(* PLC project Doqu_ges.project, CODESYS CODESYS V3.5 SP20 Patch 1 *)
(* stored: creationDateTime 2024-07-29T14:44:46.2377894, modificationDateTime 2024-07-20T22:10:28.0263958 *)

{attribute 'qualified_only'}
VAR_GLOBAL  (* GVL_1 *)
  Pry_Net_Radition_104 AT %QD10 : REAL;  (* NEW Pyronometer *)
  Pry_Compensated_Radition_104 AT %QD11 : REAL;
  Pry_Temp_104 AT %QD12 : REAL;
  Pry_External_Voltage_104 AT %QD13 : REAL;
  Refcel1_Net_Radition_104 AT %QD14 : REAL;  (* Refcel-1 *)
  Refcel1_Compensated_Radition_104 AT %QD15 : REAL;
  Refcel1_Temp_104 AT %QD16 : REAL;
  Refcel2_Net_Radition_104 AT %QD17 : REAL;  (* Refcel-2 *)
  Refcel2_Compensated_Radition_104 AT %QD18 : REAL;
  Refcel2_Temp_104 AT %QD19 : REAL;
  H1_Ia_104 AT %QD20 : REAL;  (* H1_Relay *)
  H1_Ib_104 AT %QD21 : REAL;
  H1_Ic_104 AT %QD22 : REAL;
  H1_Fault_Ia_104 AT %QD23 : REAL;
  H1_Fault_Ib_104 AT %QD24 : REAL;
  H1_Fault_Ic_104 AT %QD25 : REAL;
  H1_In_104 AT %QD26 : REAL;
  H1_Va_104 AT %QD27 : REAL;
  H1_Vb_104 AT %QD28 : REAL;
  H1_Vc_104 AT %QD29 : REAL;
  H1_Van_104 AT %QD30 : REAL;
  H1_Vbn_104 AT %QD31 : REAL;
  H1_Vcn_104 AT %QD32 : REAL;
  H1_F_104 AT %QD33 : REAL;
  H1_THD_Ia_104 AT %QD34 : REAL;
  H1_THD_Ib_104 AT %QD35 : REAL;
  H1_THD_Ic_104 AT %QD36 : REAL;
  H1_THD_Va_104 AT %QD37 : REAL;
  H1_THD_Vb_104 AT %QD38 : REAL;
  H1_THD_Vc_104 AT %QD39 : REAL;
  H1_Pf_104 AT %QD40 : REAL;
  H1_P_104 AT %QD41 : REAL;
  H1_Q_104 AT %QD42 : REAL;
  H1_S_104 AT %QD43 : REAL;
  H1_Wpneg_104 AT %QD44 : REAL;
  H1_Wqneg_104 AT %QD45 : REAL;
  H1_Wppos_104 AT %QD46 : REAL;
  H1_Wqpos_104 AT %QD47 : REAL;
  H1_CB_State_104 AT %QD48 : REAL;
  H1_DS_State_104 AT %QD49 : REAL;
  H1_EDS_State_104 AT %QD50 : REAL;
  H1_Remote_State_104 AT %QD51 : REAL;
  H1_OC_State1_104 AT %QD52 : REAL;
  H1_OC_State2_104 AT %QD53 : REAL;
  H1_EOC_State1_104 AT %QD54 : REAL;
  H1_EOC_State2_104 AT %QD55 : REAL;
  H1_Relay_Fault_104 AT %QD56 : REAL;
  H2_Ia_104 AT %QD57 : REAL;  (* H2_ION *)
  H2_Ib_104 AT %QD58 : REAL;
  H2_Ic_104 AT %QD59 : REAL;
  H2_Van_104 AT %QD60 : REAL;
  H2_Vbn_104 AT %QD61 : REAL;
  H2_Vcn_104 AT %QD62 : REAL;
  H2_Vab_104 AT %QD63 : REAL;
  H2_Vbc_104 AT %QD64 : REAL;
  H2_Vac_104 AT %QD65 : REAL;
  H2_F_104 AT %QD66 : REAL;
  H2_PF_104 AT %QD67 : REAL;
  H2_THDIA_104 AT %QD68 : REAL;
  H2_THDIB_104 AT %QD69 : REAL;
  H2_THDIC_104 AT %QD70 : REAL;
  H2_THDVA_104 AT %QD71 : REAL;
  H2_THDVB_104 AT %QD72 : REAL;
  H2_THDVC_104 AT %QD73 : REAL;
  H2_P_104 AT %QD74 : REAL;
  H2_Q_104 AT %QD75 : REAL;
  H2_S_104 AT %QD76 : REAL;
  H2_Wppos_104 AT %QD77 : REAL;
  H2_Wpneg_104 AT %QD78 : REAL;
  H2_Wqpos_104 AT %QD79 : REAL;
  H2_Wqneg_104 AT %QD80 : REAL;
  H2_Ia_Angle_104 AT %QD81 : REAL;
  H2_Ib_Angle_104 AT %QD82 : REAL;
  H2_Ic_Angle_104 AT %QD83 : REAL;
  H2_Va_Angle_104 AT %QD84 : REAL;
  H2_Vb_Angle_104 AT %QD85 : REAL;
  H2_Vc_Angle_104 AT %QD86 : REAL;
  H2_V1Plt_104 AT %QD87 : REAL;
  H2_V1Pst_104 AT %QD88 : REAL;
  H2_V2Plt_104 AT %QD89 : REAL;
  H2_V2Pst_104 AT %QD90 : REAL;
  H2_V3Plt_104 AT %QD91 : REAL;
  H2_V3Pst_104 AT %QD92 : REAL;
  INV1_Status_104 AT %QD93 : REAL;  (* *Inverter-1 *)
  INV1_Status_1044 : REAL;
  INV1_Pin_104 AT %QD94 : REAL;
  INV1_Pv1_voltage_104 AT %QD95 : REAL;
  INV1_Pv1_current_104 AT %QD96 : REAL;
  INV1_Pv1_Pin_104 AT %QD97 : REAL;
  INV1_Pv2_voltage_104 AT %QD98 : REAL;
  INV1_Pv2_current_104 AT %QD99 : REAL;
  INV1_Pv2_Pin_104 AT %QD100 : REAL;
  INV1_Pv3_voltage_104 AT %QD101 : REAL;
  INV1_Pv3_current_104 AT %QD102 : REAL;
  INV1_Pv3_Pin_104 AT %QD103 : REAL;
  INV1_Pv4_voltage_104 AT %QD104 : REAL;
  INV1_Pv4_current_104 AT %QD105 : REAL;
  INV1_Pv4_Pin_104 AT %QD106 : REAL;
  INV1_Pv5_voltage_104 AT %QD107 : REAL;
  INV1_Pv5_current_104 AT %QD108 : REAL;
  INV1_Pv5_Pin_104 AT %QD109 : REAL;
  INV1_Pv6_voltage_104 AT %QD110 : REAL;
  INV1_Pv6_current_104 AT %QD111 : REAL;
  INV1_Pv6_Pin_104 AT %QD112 : REAL;
  INV1_Pv7_voltage_104 AT %QD113 : REAL;
  INV1_Pv7_current_104 AT %QD114 : REAL;
  INV1_Pv7_Pin_104 AT %QD115 : REAL;
  INV1_Pv8_voltage_104 AT %QD116 : REAL;
  INV1_Pv8_current_104 AT %QD117 : REAL;
  INV1_Pv8_Pin_104 AT %QD118 : REAL;
  INV1_Pv9_voltage_104 AT %QD119 : REAL;
  INV1_Pv9_current_104 AT %QD120 : REAL;
  INV1_Pv9_Pin_104 AT %QD121 : REAL;
  INV1_Pv10_voltage_104 AT %QD122 : REAL;
  INV1_Pv10_current_104 AT %QD123 : REAL;
  INV1_Pv10_Pin_104 AT %QD124 : REAL;
  INV1_Pac_out_104 AT %QD125 : REAL;
  INV1_Fac_104 AT %QD126 : REAL;
  INV1_Vac1_104 AT %QD127 : REAL;
  INV1_Iac1_104 AT %QD128 : REAL;
  INV1_Pac1_104 AT %QD129 : REAL;
  INV1_Vac2_104 AT %QD130 : REAL;
  INV1_Iac2_104 AT %QD131 : REAL;
  INV1_Pac2_104 AT %QD132 : REAL;
  INV1_Vac3_104 AT %QD133 : REAL;
  INV1_Iac3_104 AT %QD134 : REAL;
  INV1_Pac3_104 AT %QD135 : REAL;
  INV1_Vac_RS_104 AT %QD136 : REAL;
  INV1_Vac_ST_104 AT %QD137 : REAL;
  INV1_Vac_TR_104 AT %QD138 : REAL;
  INV1_Eactoday_104 AT %QD139 : REAL;
  INV1_Eactotal_104 AT %QD140 : REAL;
  INV1_Timetotal_104 AT %QD141 : REAL;
  INV1_Epv1_today_104 AT %QD142 : REAL;
  INV1_Epv1_total_104 AT %QD143 : REAL;
  INV1_Epv2_today_104 AT %QD144 : REAL;
  INV1_Epv2_total_104 AT %QD145 : REAL;
  INV1_Epv3_today_104 AT %QD146 : REAL;
  INV1_Epv3_total_104 AT %QD147 : REAL;
  INV1_Epv4_today_104 AT %QD148 : REAL;
  INV1_Epv4_total_104 AT %QD149 : REAL;
  INV1_Epv5_today_104 AT %QD150 : REAL;
  INV1_Epv5_total_104 AT %QD151 : REAL;
  INV1_Epv6_today_104 AT %QD152 : REAL;
  INV1_Epv6_total_104 AT %QD153 : REAL;
  INV1_Epv7_today_104 AT %QD154 : REAL;
  INV1_Epv7_total_104 AT %QD155 : REAL;
  INV1_Epv8_today_104 AT %QD156 : REAL;
  INV1_Epv8_total_104 AT %QD157 : REAL;
  INV1_Epv9_today_104 AT %QD158 : REAL;
  INV1_Epv9_total_104 AT %QD159 : REAL;
  INV1_Epv10_today_104 AT %QD160 : REAL;
  INV1_Epv10_total_104 AT %QD161 : REAL;
  INV1_Epv_total_104 AT %QD162 : REAL;
  INV1_Temp1_104 AT %QD163 : REAL;
  INV1_Temp2_104 AT %QD164 : REAL;
  INV1_Temp3_104 AT %QD165 : REAL;
  INV1_Temp4_104 AT %QD166 : REAL;
  INV1_BatVolt_DSP_104 AT %QD167 : REAL;
  INV1_P_Bus_Voltage_104 AT %QD168 : REAL;
  INV1_N_Bus_Voltage_104 AT %QD169 : REAL;
  INV1_IPF_104 AT %QD170 : REAL;
  INV1_String_V1_104 AT %QD171 : REAL;
  INV1_String_I1_104 AT %QD172 : REAL;
  INV1_String_V2_104 AT %QD173 : REAL;
  INV1_String_I2_104 AT %QD174 : REAL;
  INV1_String_V3_104 AT %QD175 : REAL;
  INV1_String_I3_104 AT %QD176 : REAL;
  INV1_String_V4_104 AT %QD177 : REAL;
  INV1_String_I4_104 AT %QD178 : REAL;
  INV1_String_V5_104 AT %QD179 : REAL;
  INV1_String_I5_104 AT %QD180 : REAL;
  INV1_String_V6_104 AT %QD181 : REAL;
  INV1_String_I6_104 AT %QD182 : REAL;
  INV1_String_V7_104 AT %QD183 : REAL;
  INV1_String_I7_104 AT %QD184 : REAL;
  INV1_String_V8_104 AT %QD185 : REAL;
  INV1_String_I8_104 AT %QD186 : REAL;
  INV1_String_V9_104 AT %QD187 : REAL;
  INV1_String_I9_104 AT %QD188 : REAL;
  INV1_String_V10_104 AT %QD189 : REAL;
  INV1_String_I10_104 AT %QD190 : REAL;
  INV1_String_V11_104 AT %QD191 : REAL;
  INV1_String_I11_104 AT %QD192 : REAL;
  INV1_String_V12_104 AT %QD193 : REAL;
  INV1_String_I12_104 AT %QD194 : REAL;
  INV1_String_V13_104 AT %QD195 : REAL;
  INV1_String_I13_104 AT %QD196 : REAL;
  INV1_String_V14_104 AT %QD197 : REAL;
  INV1_String_I14_104 AT %QD198 : REAL;
  INV1_String_V15_104 AT %QD199 : REAL;
  INV1_String_I15_104 AT %QD200 : REAL;
  INV1_String_V16_104 AT %QD201 : REAL;
  INV1_String_I16_104 AT %QD202 : REAL;
  INV1_String_V17_104 AT %QD203 : REAL;
  INV1_String_I17_104 AT %QD204 : REAL;
  INV1_String_V18_104 AT %QD205 : REAL;
  INV1_String_I18_104 AT %QD206 : REAL;
  INV1_String_V19_104 AT %QD207 : REAL;
  INV1_String_I19_104 AT %QD208 : REAL;
  INV1_String_V20_104 AT %QD209 : REAL;
  INV1_String_I20_104 AT %QD210 : REAL;
  INV1_Fan1_Fault_104 AT %QD211 : REAL;
  INV1_Fan2_Fault_104 AT %QD212 : REAL;
  INV1_Fan3_Fault_104 AT %QD213 : REAL;
  INV1_Fan4_Fault_104 AT %QD214 : REAL;
  INV2_Status_104 AT %QD215 : REAL;  (* Inverter-2 *)
  INV2_Pin_104 AT %QD216 : REAL;
  INV2_Pv1_voltage_104 AT %QD217 : REAL;
  INV2_Pv1_current_104 AT %QD218 : REAL;
  INV2_Pv1_Pin_104 AT %QD219 : REAL;
  INV2_Pv2_voltage_104 AT %QD220 : REAL;
  INV2_Pv2_current_104 AT %QD221 : REAL;
  INV2_Pv2_Pin_104 AT %QD222 : REAL;
  INV2_Pv3_voltage_104 AT %QD223 : REAL;
  INV2_Pv3_current_104 AT %QD224 : REAL;
  INV2_Pv3_Pin_104 AT %QD225 : REAL;
  INV2_Pv4_voltage_104 AT %QD226 : REAL;
  INV2_Pv4_current_104 AT %QD227 : REAL;
  INV2_Pv4_Pin_104 AT %QD228 : REAL;
  INV2_Pv5_voltage_104 AT %QD229 : REAL;
  INV2_Pv5_current_104 AT %QD230 : REAL;
  INV2_Pv5_Pin_104 AT %QD231 : REAL;
  INV2_Pv6_voltage_104 AT %QD232 : REAL;
  INV2_Pv6_current_104 AT %QD233 : REAL;
  INV2_Pv6_Pin_104 AT %QD234 : REAL;
  INV2_Pv7_voltage_104 AT %QD235 : REAL;
  INV2_Pv7_current_104 AT %QD236 : REAL;
  INV2_Pv7_Pin_104 AT %QD237 : REAL;
  INV2_Pv8_voltage_104 AT %QD238 : REAL;
  INV2_Pv8_current_104 AT %QD239 : REAL;
  INV2_Pv8_Pin_104 AT %QD240 : REAL;
  INV2_Pv9_voltage_104 AT %QD241 : REAL;
  INV2_Pv9_current_104 AT %QD242 : REAL;
  INV2_Pv9_Pin_104 AT %QD243 : REAL;
  INV2_Pv10_voltage_104 AT %QD244 : REAL;
  INV2_Pv10_current_104 AT %QD245 : REAL;
  INV2_Pv10_Pin_104 AT %QD246 : REAL;
  INV2_Pac_out_104 AT %QD247 : REAL;
  INV2_Fac_104 AT %QD248 : REAL;
  INV2_Vac1_104 AT %QD249 : REAL;
  INV2_Iac1_104 AT %QD250 : REAL;
  INV2_Pac1_104 AT %QD251 : REAL;
  INV2_Vac2_104 AT %QD252 : REAL;
  INV2_Iac2_104 AT %QD253 : REAL;
  INV2_Pac2_104 AT %QD254 : REAL;
  INV2_Vac3_104 AT %QD255 : REAL;
  INV2_Iac3_104 AT %QD256 : REAL;
  INV2_Pac3_104 AT %QD257 : REAL;
  INV2_Vac_RS_104 AT %QD258 : REAL;
  INV2_Vac_ST_104 AT %QD259 : REAL;
  INV2_Vac_TR_104 AT %QD260 : REAL;
  INV2_Eactoday_104 AT %QD261 : REAL;
  INV2_Eactotal_104 AT %QD262 : REAL;
  INV2_Timetotal_104 AT %QD263 : REAL;
  INV2_Epv1_today_104 AT %QD264 : REAL;
  INV2_Epv1_total_104 AT %QD265 : REAL;
  INV2_Epv2_today_104 AT %QD266 : REAL;
  INV2_Epv2_total_104 AT %QD267 : REAL;
  INV2_Epv3_today_104 AT %QD268 : REAL;
  INV2_Epv3_total_104 AT %QD269 : REAL;
  INV2_Epv4_today_104 AT %QD270 : REAL;
  INV2_Epv4_total_104 AT %QD271 : REAL;
  INV2_Epv5_today_104 AT %QD272 : REAL;
  INV2_Epv5_total_104 AT %QD273 : REAL;
  INV2_Epv6_today_104 AT %QD274 : REAL;
  INV2_Epv6_total_104 AT %QD275 : REAL;
  INV2_Epv7_today_104 AT %QD276 : REAL;
  INV2_Epv7_total_104 AT %QD277 : REAL;
  INV2_Epv8_today_104 AT %QD278 : REAL;
  INV2_Epv8_total_104 AT %QD279 : REAL;
  INV2_Epv9_today_104 AT %QD280 : REAL;
  INV2_Epv9_total_104 AT %QD281 : REAL;
  INV2_Epv10_today_104 AT %QD282 : REAL;
  INV2_Epv10_total_104 AT %QD283 : REAL;
  INV2_Epv_total_104 AT %QD284 : REAL;
  INV2_Temp1_104 AT %QD285 : REAL;
  INV2_Temp2_104 AT %QD286 : REAL;
  INV2_Temp3_104 AT %QD287 : REAL;
  INV2_Temp4_104 AT %QD288 : REAL;
  INV2_BatVolt_DSP_104 AT %QD289 : REAL;
  INV2_P_Bus_Voltage_104 AT %QD290 : REAL;
  INV2_N_Bus_Voltage_104 AT %QD291 : REAL;
  INV2_IPF_104 AT %QD292 : REAL;
  INV2_String_V1_104 AT %QD293 : REAL;
  INV2_String_I1_104 AT %QD294 : REAL;
  INV2_String_V2_104 AT %QD295 : REAL;
  INV2_String_I2_104 AT %QD296 : REAL;
  INV2_String_V3_104 AT %QD297 : REAL;
  INV2_String_I3_104 AT %QD298 : REAL;
  INV2_String_V4_104 AT %QD299 : REAL;
  INV2_String_I4_104 AT %QD300 : REAL;
  INV2_String_V5_104 AT %QD301 : REAL;
  INV2_String_I5_104 AT %QD302 : REAL;
  INV2_String_V6_104 AT %QD303 : REAL;
  INV2_String_I6_104 AT %QD304 : REAL;
  INV2_String_V7_104 AT %QD305 : REAL;
  INV2_String_I7_104 AT %QD306 : REAL;
  INV2_String_V8_104 AT %QD307 : REAL;
  INV2_String_I8_104 AT %QD308 : REAL;
  INV2_String_V9_104 AT %QD309 : REAL;
  INV2_String_I9_104 AT %QD310 : REAL;
  INV2_String_V10_104 AT %QD311 : REAL;
  INV2_String_I10_104 AT %QD312 : REAL;
  INV2_String_V11_104 AT %QD313 : REAL;
  INV2_String_I11_104 AT %QD314 : REAL;
  INV2_String_V12_104 AT %QD315 : REAL;
  INV2_String_I12_104 AT %QD316 : REAL;
  INV2_String_V13_104 AT %QD317 : REAL;
  INV2_String_I13_104 AT %QD318 : REAL;
  INV2_String_V14_104 AT %QD319 : REAL;
  INV2_String_I14_104 AT %QD320 : REAL;
  INV2_String_V15_104 AT %QD321 : REAL;
  INV2_String_I15_104 AT %QD322 : REAL;
  INV2_String_V16_104 AT %QD323 : REAL;
  INV2_String_I16_104 AT %QD324 : REAL;
  INV2_String_V17_104 AT %QD325 : REAL;
  INV2_String_I17_104 AT %QD326 : REAL;
  INV2_String_V18_104 AT %QD327 : REAL;
  INV2_String_I18_104 AT %QD328 : REAL;
  INV2_String_V19_104 AT %QD329 : REAL;
  INV2_String_I19_104 AT %QD330 : REAL;
  INV2_String_V20_104 AT %QD331 : REAL;
  INV2_String_I20_104 AT %QD332 : REAL;
  INV2_Fan1_Fault_104 AT %QD333 : REAL;
  INV2_Fan2_Fault_104 AT %QD334 : REAL;
  INV2_Fan3_Fault_104 AT %QD335 : REAL;
  INV2_Fan4_Fault_104 AT %QD336 : REAL;
  INV3_Status_104 AT %QD337 : REAL;  (* *Inverter-3* *)
  INV3_Pin_104 AT %QD338 : REAL;
  INV3_Pv1_voltage_104 AT %QD339 : REAL;
  INV3_Pv1_current_104 AT %QD340 : REAL;
  INV3_Pv1_Pin_104 AT %QD341 : REAL;
  INV3_Pv2_voltage_104 AT %QD342 : REAL;
  INV3_Pv2_current_104 AT %QD343 : REAL;
  INV3_Pv2_Pin_104 AT %QD344 : REAL;
  INV3_Pv3_voltage_104 AT %QD345 : REAL;
  INV3_Pv3_current_104 AT %QD346 : REAL;
  INV3_Pv3_Pin_104 AT %QD347 : REAL;
  INV3_Pv4_voltage_104 AT %QD348 : REAL;
  INV3_Pv4_current_104 AT %QD349 : REAL;
  INV3_Pv4_Pin_104 AT %QD350 : REAL;
  INV3_Pv5_voltage_104 AT %QD351 : REAL;
  INV3_Pv5_current_104 AT %QD352 : REAL;
  INV3_Pv5_Pin_104 AT %QD353 : REAL;
  INV3_Pv6_voltage_104 AT %QD354 : REAL;
  INV3_Pv6_current_104 AT %QD355 : REAL;
  INV3_Pv6_Pin_104 AT %QD356 : REAL;
  INV3_Pv7_voltage_104 AT %QD357 : REAL;
  INV3_Pv7_current_104 AT %QD358 : REAL;
  INV3_Pv7_Pin_104 AT %QD359 : REAL;
  INV3_Pv8_voltage_104 AT %QD360 : REAL;
  INV3_Pv8_current_104 AT %QD361 : REAL;
  INV3_Pv8_Pin_104 AT %QD362 : REAL;
  INV3_Pv9_voltage_104 AT %QD363 : REAL;
  INV3_Pv9_current_104 AT %QD364 : REAL;
  INV3_Pv9_Pin_104 AT %QD365 : REAL;
  INV3_Pv10_voltage_104 AT %QD366 : REAL;
  INV3_Pv10_current_104 AT %QD367 : REAL;
  INV3_Pv10_Pin_104 AT %QD368 : REAL;
  INV3_Pac_out_104 AT %QD369 : REAL;
  INV3_Fac_104 AT %QD370 : REAL;
  INV3_Vac1_104 AT %QD371 : REAL;
  INV3_Iac1_104 AT %QD372 : REAL;
  INV3_Pac1_104 AT %QD373 : REAL;
  INV3_Vac2_104 AT %QD374 : REAL;
  INV3_Iac2_104 AT %QD375 : REAL;
  INV3_Pac2_104 AT %QD376 : REAL;
  INV3_Vac3_104 AT %QD377 : REAL;
  INV3_Iac3_104 AT %QD378 : REAL;
  INV3_Pac3_104 AT %QD379 : REAL;
  INV3_Vac_RS_104 AT %QD380 : REAL;
  INV3_Vac_ST_104 AT %QD381 : REAL;
  INV3_Vac_TR_104 AT %QD382 : REAL;
  INV3_Eactoday_104 AT %QD383 : REAL;
  INV3_Eactotal_104 AT %QD384 : REAL;
  INV3_Timetotal_104 AT %QD385 : REAL;
  INV3_Epv1_today_104 AT %QD386 : REAL;
  INV3_Epv1_total_104 AT %QD387 : REAL;
  INV3_Epv2_today_104 AT %QD388 : REAL;
  INV3_Epv2_total_104 AT %QD389 : REAL;
  INV3_Epv3_today_104 AT %QD390 : REAL;
  INV3_Epv3_total_104 AT %QD391 : REAL;
  INV3_Epv4_today_104 AT %QD392 : REAL;
  INV3_Epv4_total_104 AT %QD393 : REAL;
  INV3_Epv5_today_104 AT %QD394 : REAL;
  INV3_Epv5_total_104 AT %QD395 : REAL;
  INV3_Epv6_today_104 AT %QD396 : REAL;
  INV3_Epv6_total_104 AT %QD397 : REAL;
  INV3_Epv7_today_104 AT %QD398 : REAL;
  INV3_Epv7_total_104 AT %QD399 : REAL;
  INV3_Epv8_today_104 AT %QD400 : REAL;
  INV3_Epv8_total_104 AT %QD401 : REAL;
  INV3_Epv9_today_104 AT %QD402 : REAL;
  INV3_Epv9_total_104 AT %QD403 : REAL;
  INV3_Epv10_today_104 AT %QD404 : REAL;
  INV3_Epv10_total_104 AT %QD405 : REAL;
  INV3_Epv_total_104 AT %QD406 : REAL;
  INV3_Temp1_104 AT %QD407 : REAL;
  INV3_Temp2_104 AT %QD408 : REAL;
  INV3_Temp3_104 AT %QD409 : REAL;
  INV3_Temp4_104 AT %QD410 : REAL;
  INV3_BatVolt_DSP_104 AT %QD411 : REAL;
  INV3_P_Bus_Voltage_104 AT %QD412 : REAL;
  INV3_N_Bus_Voltage_104 AT %QD413 : REAL;
  INV3_IPF_104 AT %QD414 : REAL;
  INV3_String_V1_104 AT %QD415 : REAL;
  INV3_String_I1_104 AT %QD416 : REAL;
  INV3_String_V2_104 AT %QD417 : REAL;
  INV3_String_I2_104 AT %QD418 : REAL;
  INV3_String_V3_104 AT %QD419 : REAL;
  INV3_String_I3_104 AT %QD420 : REAL;
  INV3_String_V4_104 AT %QD421 : REAL;
  INV3_String_I4_104 AT %QD422 : REAL;
  INV3_String_V5_104 AT %QD423 : REAL;
  INV3_String_I5_104 AT %QD424 : REAL;
  INV3_String_V6_104 AT %QD425 : REAL;
  INV3_String_I6_104 AT %QD426 : REAL;
  INV3_String_V7_104 AT %QD427 : REAL;
  INV3_String_I7_104 AT %QD428 : REAL;
  INV3_String_V8_104 AT %QD429 : REAL;
  INV3_String_I8_104 AT %QD430 : REAL;
  INV3_String_V9_104 AT %QD431 : REAL;
  INV3_String_I9_104 AT %QD432 : REAL;
  INV3_String_V10_104 AT %QD433 : REAL;
  INV3_String_I10_104 AT %QD434 : REAL;
  INV3_String_V11_104 AT %QD435 : REAL;
  INV3_String_I11_104 AT %QD436 : REAL;
  INV3_String_V12_104 AT %QD437 : REAL;
  INV3_String_I12_104 AT %QD438 : REAL;
  INV3_String_V13_104 AT %QD439 : REAL;
  INV3_String_I13_104 AT %QD440 : REAL;
  INV3_String_V14_104 AT %QD441 : REAL;
  INV3_String_I14_104 AT %QD442 : REAL;
  INV3_String_V15_104 AT %QD443 : REAL;
  INV3_String_I15_104 AT %QD444 : REAL;
  INV3_String_V16_104 AT %QD445 : REAL;
  INV3_String_I16_104 AT %QD446 : REAL;
  INV3_String_V17_104 AT %QD447 : REAL;
  INV3_String_I17_104 AT %QD448 : REAL;
  INV3_String_V18_104 AT %QD449 : REAL;
  INV3_String_I18_104 AT %QD450 : REAL;
  INV3_String_V19_104 AT %QD451 : REAL;
  INV3_String_I19_104 AT %QD452 : REAL;
  INV3_String_V20_104 AT %QD453 : REAL;
  INV3_String_I20_104 AT %QD454 : REAL;
  INV3_Fan1_Fault_104 AT %QD455 : REAL;
  INV3_Fan2_Fault_104 AT %QD456 : REAL;
  INV3_Fan3_Fault_104 AT %QD457 : REAL;
  INV3_Fan4_Fault_104 AT %QD458 : REAL;
  INV4_Status_104 AT %QD459 : REAL;  (* *Inverter-4* *)
  INV4_Pin_104 AT %QD460 : REAL;
  INV4_Pv1_voltage_104 AT %QD461 : REAL;
  INV4_Pv1_current_104 AT %QD462 : REAL;
  INV4_Pv1_Pin_104 AT %QD463 : REAL;
  INV4_Pv2_voltage_104 AT %QD464 : REAL;
  INV4_Pv2_current_104 AT %QD465 : REAL;
  INV4_Pv2_Pin_104 AT %QD466 : REAL;
  INV4_Pv3_voltage_104 AT %QD467 : REAL;
  INV4_Pv3_current_104 AT %QD468 : REAL;
  INV4_Pv3_Pin_104 AT %QD469 : REAL;
  INV4_Pv4_voltage_104 AT %QD470 : REAL;
  INV4_Pv4_current_104 AT %QD471 : REAL;
  INV4_Pv4_Pin_104 AT %QD472 : REAL;
  INV4_Pv5_voltage_104 AT %QD473 : REAL;
  INV4_Pv5_current_104 AT %QD474 : REAL;
  INV4_Pv5_Pin_104 AT %QD475 : REAL;
  INV4_Pv6_voltage_104 AT %QD476 : REAL;
  INV4_Pv6_current_104 AT %QD477 : REAL;
  INV4_Pv6_Pin_104 AT %QD478 : REAL;
  INV4_Pv7_voltage_104 AT %QD479 : REAL;
  INV4_Pv7_current_104 AT %QD480 : REAL;
  INV4_Pv7_Pin_104 AT %QD481 : REAL;
  INV4_Pv8_voltage_104 AT %QD482 : REAL;
  INV4_Pv8_current_104 AT %QD483 : REAL;
  INV4_Pv8_Pin_104 AT %QD484 : REAL;
  INV4_Pv9_voltage_104 AT %QD485 : REAL;
  INV4_Pv9_current_104 AT %QD486 : REAL;
  INV4_Pv9_Pin_104 AT %QD487 : REAL;
  INV4_Pv10_voltage_104 AT %QD488 : REAL;
  INV4_Pv10_current_104 AT %QD489 : REAL;
  INV4_Pv10_Pin_104 AT %QD490 : REAL;
  INV4_Pac_out_104 AT %QD491 : REAL;
  INV4_Fac_104 AT %QD492 : REAL;
  INV4_Vac1_104 AT %QD493 : REAL;
  INV4_Iac1_104 AT %QD494 : REAL;
  INV4_Pac1_104 AT %QD495 : REAL;
  INV4_Vac2_104 AT %QD496 : REAL;
  INV4_Iac2_104 AT %QD497 : REAL;
  INV4_Pac2_104 AT %QD498 : REAL;
  INV4_Vac3_104 AT %QD499 : REAL;
  INV4_Iac3_104 AT %QD500 : REAL;
  INV4_Pac3_104 AT %QD501 : REAL;
  INV4_Vac_RS_104 AT %QD502 : REAL;
  INV4_Vac_ST_104 AT %QD503 : REAL;
  INV4_Vac_TR_104 AT %QD504 : REAL;
  INV4_Eactoday_104 AT %QD505 : REAL;
  INV4_Eactotal_104 AT %QD506 : REAL;
  INV4_Timetotal_104 AT %QD507 : REAL;
  INV4_Epv1_today_104 AT %QD508 : REAL;
  INV4_Epv1_total_104 AT %QD509 : REAL;
  INV4_Epv2_today_104 AT %QD510 : REAL;
  INV4_Epv2_total_104 AT %QD511 : REAL;
  INV4_Epv3_today_104 AT %QD512 : REAL;
  INV4_Epv3_total_104 AT %QD513 : REAL;
  INV4_Epv4_today_104 AT %QD514 : REAL;
  INV4_Epv4_total_104 AT %QD515 : REAL;
  INV4_Epv5_today_104 AT %QD516 : REAL;
  INV4_Epv5_total_104 AT %QD517 : REAL;
  INV4_Epv6_today_104 AT %QD518 : REAL;
  INV4_Epv6_total_104 AT %QD519 : REAL;
  INV4_Epv7_today_104 AT %QD520 : REAL;
  INV4_Epv7_total_104 AT %QD521 : REAL;
  INV4_Epv8_today_104 AT %QD522 : REAL;
  INV4_Epv8_total_104 AT %QD523 : REAL;
  INV4_Epv9_today_104 AT %QD524 : REAL;
  INV4_Epv9_total_104 AT %QD525 : REAL;
  INV4_Epv10_today_104 AT %QD526 : REAL;
  INV4_Epv10_total_104 AT %QD527 : REAL;
  INV4_Epv_total_104 AT %QD528 : REAL;
  INV4_Temp1_104 AT %QD529 : REAL;
  INV4_Temp2_104 AT %QD530 : REAL;
  INV4_Temp3_104 AT %QD531 : REAL;
  INV4_Temp4_104 AT %QD532 : REAL;
  INV4_BatVolt_DSP_104 AT %QD533 : REAL;
  INV4_P_Bus_Voltage_104 AT %QD534 : REAL;
  INV4_N_Bus_Voltage_104 AT %QD535 : REAL;
  INV4_IPF_104 AT %QD536 : REAL;
  INV4_String_V1_104 AT %QD537 : REAL;
  INV4_String_I1_104 AT %QD538 : REAL;
  INV4_String_V2_104 AT %QD539 : REAL;
  INV4_String_I2_104 AT %QD540 : REAL;
  INV4_String_V3_104 AT %QD541 : REAL;
  INV4_String_I3_104 AT %QD542 : REAL;
  INV4_String_V4_104 AT %QD543 : REAL;
  INV4_String_I4_104 AT %QD544 : REAL;
  INV4_String_V5_104 AT %QD545 : REAL;
  INV4_String_I5_104 AT %QD546 : REAL;
  INV4_String_V6_104 AT %QD547 : REAL;
  INV4_String_I6_104 AT %QD548 : REAL;
  INV4_String_V7_104 AT %QD549 : REAL;
  INV4_String_I7_104 AT %QD550 : REAL;
  INV4_String_V8_104 AT %QD551 : REAL;
  INV4_String_I8_104 AT %QD552 : REAL;
  INV4_String_V9_104 AT %QD553 : REAL;
  INV4_String_I9_104 AT %QD554 : REAL;
  INV4_String_V10_104 AT %QD555 : REAL;
  INV4_String_I10_104 AT %QD556 : REAL;
  INV4_String_V11_104 AT %QD557 : REAL;
  INV4_String_I11_104 AT %QD558 : REAL;
  INV4_String_V12_104 AT %QD559 : REAL;
  INV4_String_I12_104 AT %QD560 : REAL;
  INV4_String_V13_104 AT %QD561 : REAL;
  INV4_String_I13_104 AT %QD562 : REAL;
  INV4_String_V14_104 AT %QD563 : REAL;
  INV4_String_I14_104 AT %QD564 : REAL;
  INV4_String_V15_104 AT %QD565 : REAL;
  INV4_String_I15_104 AT %QD566 : REAL;
  INV4_String_V16_104 AT %QD567 : REAL;
  INV4_String_I16_104 AT %QD568 : REAL;
  INV4_String_V17_104 AT %QD569 : REAL;
  INV4_String_I17_104 AT %QD570 : REAL;
  INV4_String_V18_104 AT %QD571 : REAL;
  INV4_String_I18_104 AT %QD572 : REAL;
  INV4_String_V19_104 AT %QD573 : REAL;
  INV4_String_I19_104 AT %QD574 : REAL;
  INV4_String_V20_104 AT %QD575 : REAL;
  INV4_String_I20_104 AT %QD576 : REAL;
  INV4_Fan1_Fault_104 AT %QD577 : REAL;
  INV4_Fan2_Fault_104 AT %QD578 : REAL;
  INV4_Fan3_Fault_104 AT %QD579 : REAL;
  INV4_Fan4_Fault_104 AT %QD580 : REAL;
  INV5_Status_104 AT %QD581 : REAL;  (* *Inverter-5* *)
  INV5_Pin_104 AT %QD582 : REAL;
  INV5_Pv1_voltage_104 AT %QD583 : REAL;
  INV5_Pv1_current_104 AT %QD584 : REAL;
  INV5_Pv1_Pin_104 AT %QD585 : REAL;
  INV5_Pv2_voltage_104 AT %QD586 : REAL;
  INV5_Pv2_current_104 AT %QD587 : REAL;
  INV5_Pv2_Pin_104 AT %QD588 : REAL;
  INV5_Pv3_voltage_104 AT %QD589 : REAL;
  INV5_Pv3_current_104 AT %QD590 : REAL;
  INV5_Pv3_Pin_104 AT %QD591 : REAL;
  INV5_Pv4_voltage_104 AT %QD592 : REAL;
  INV5_Pv4_current_104 AT %QD593 : REAL;
  INV5_Pv4_Pin_104 AT %QD594 : REAL;
  INV5_Pv5_voltage_104 AT %QD595 : REAL;
  INV5_Pv5_current_104 AT %QD596 : REAL;
  INV5_Pv5_Pin_104 AT %QD597 : REAL;
  INV5_Pv6_voltage_104 AT %QD598 : REAL;
  INV5_Pv6_current_104 AT %QD599 : REAL;
  INV5_Pv6_Pin_104 AT %QD600 : REAL;
  INV5_Pv7_voltage_104 AT %QD601 : REAL;
  INV5_Pv7_current_104 AT %QD602 : REAL;
  INV5_Pv7_Pin_104 AT %QD603 : REAL;
  INV5_Pv8_voltage_104 AT %QD604 : REAL;
  INV5_Pv8_current_104 AT %QD605 : REAL;
  INV5_Pv8_Pin_104 AT %QD606 : REAL;
  INV5_Pv9_voltage_104 AT %QD607 : REAL;
  INV5_Pv9_current_104 AT %QD608 : REAL;
  INV5_Pv9_Pin_104 AT %QD609 : REAL;
  INV5_Pv10_voltage_104 AT %QD610 : REAL;
  INV5_Pv10_current_104 AT %QD611 : REAL;
  INV5_Pv10_Pin_104 AT %QD612 : REAL;
  INV5_Pac_out_104 AT %QD613 : REAL;
  INV5_Fac_104 AT %QD614 : REAL;
  INV5_Vac1_104 AT %QD615 : REAL;
  INV5_Iac1_104 AT %QD616 : REAL;
  INV5_Pac1_104 AT %QD617 : REAL;
  INV5_Vac2_104 AT %QD618 : REAL;
  INV5_Iac2_104 AT %QD619 : REAL;
  INV5_Pac2_104 AT %QD620 : REAL;
  INV5_Vac3_104 AT %QD621 : REAL;
  INV5_Iac3_104 AT %QD622 : REAL;
  INV5_Pac3_104 AT %QD623 : REAL;
  INV5_Vac_RS_104 AT %QD624 : REAL;
  INV5_Vac_ST_104 AT %QD625 : REAL;
  INV5_Vac_TR_104 AT %QD626 : REAL;
  INV5_Eactoday_104 AT %QD627 : REAL;
  INV5_Eactotal_104 AT %QD628 : REAL;
  INV5_Timetotal_104 AT %QD629 : REAL;
  INV5_Epv1_today_104 AT %QD630 : REAL;
  INV5_Epv1_total_104 AT %QD631 : REAL;
  INV5_Epv2_today_104 AT %QD632 : REAL;
  INV5_Epv2_total_104 AT %QD633 : REAL;
  INV5_Epv3_today_104 AT %QD634 : REAL;
  INV5_Epv3_total_104 AT %QD635 : REAL;
  INV5_Epv4_today_104 AT %QD636 : REAL;
  INV5_Epv4_total_104 AT %QD637 : REAL;
  INV5_Epv5_today_104 AT %QD638 : REAL;
  INV5_Epv5_total_104 AT %QD639 : REAL;
  INV5_Epv6_today_104 AT %QD640 : REAL;
  INV5_Epv6_total_104 AT %QD641 : REAL;
  INV5_Epv7_today_104 AT %QD642 : REAL;
  INV5_Epv7_total_104 AT %QD643 : REAL;
  INV5_Epv8_today_104 AT %QD644 : REAL;
  INV5_Epv8_total_104 AT %QD645 : REAL;
  INV5_Epv9_today_104 AT %QD646 : REAL;
  INV5_Epv9_total_104 AT %QD647 : REAL;
  INV5_Epv10_today_104 AT %QD648 : REAL;
  INV5_Epv10_total_104 AT %QD649 : REAL;
  INV5_Epv_total_104 AT %QD650 : REAL;
  INV5_Temp1_104 AT %QD651 : REAL;
  INV5_Temp2_104 AT %QD652 : REAL;
  INV5_Temp3_104 AT %QD653 : REAL;
  INV5_Temp4_104 AT %QD654 : REAL;
  INV5_BatVolt_DSP_104 AT %QD655 : REAL;
  INV5_P_Bus_Voltage_104 AT %QD656 : REAL;
  INV5_N_Bus_Voltage_104 AT %QD657 : REAL;
  INV5_IPF_104 AT %QD658 : REAL;
  INV5_String_V1_104 AT %QD659 : REAL;
  INV5_String_I1_104 AT %QD660 : REAL;
  INV5_String_V2_104 AT %QD661 : REAL;
  INV5_String_I2_104 AT %QD662 : REAL;
  INV5_String_V3_104 AT %QD663 : REAL;
  INV5_String_I3_104 AT %QD664 : REAL;
  INV5_String_V4_104 AT %QD665 : REAL;
  INV5_String_I4_104 AT %QD666 : REAL;
  INV5_String_V5_104 AT %QD667 : REAL;
  INV5_String_I5_104 AT %QD668 : REAL;
  INV5_String_V6_104 AT %QD669 : REAL;
  INV5_String_I6_104 AT %QD670 : REAL;
  INV5_String_V7_104 AT %QD671 : REAL;
  INV5_String_I7_104 AT %QD672 : REAL;
  INV5_String_V8_104 AT %QD673 : REAL;
  INV5_String_I8_104 AT %QD674 : REAL;
  INV5_String_V9_104 AT %QD675 : REAL;
  INV5_String_I9_104 AT %QD676 : REAL;
  INV5_String_V10_104 AT %QD677 : REAL;
  INV5_String_I10_104 AT %QD678 : REAL;
  INV5_String_V11_104 AT %QD679 : REAL;
  INV5_String_I11_104 AT %QD680 : REAL;
  INV5_String_V12_104 AT %QD681 : REAL;
  INV5_String_I12_104 AT %QD682 : REAL;
  INV5_String_V13_104 AT %QD683 : REAL;
  INV5_String_I13_104 AT %QD684 : REAL;
  INV5_String_V14_104 AT %QD685 : REAL;
  INV5_String_I14_104 AT %QD686 : REAL;
  INV5_String_V15_104 AT %QD687 : REAL;
  INV5_String_I15_104 AT %QD688 : REAL;
  INV5_String_V16_104 AT %QD689 : REAL;
  INV5_String_I16_104 AT %QD690 : REAL;
  INV5_String_V17_104 AT %QD691 : REAL;
  INV5_String_I17_104 AT %QD692 : REAL;
  INV5_String_V18_104 AT %QD693 : REAL;
  INV5_String_I18_104 AT %QD694 : REAL;
  INV5_String_V19_104 AT %QD695 : REAL;
  INV5_String_I19_104 AT %QD696 : REAL;
  INV5_String_V20_104 AT %QD697 : REAL;
  INV5_String_I20_104 AT %QD698 : REAL;
  INV5_Fan1_Fault_104 AT %QD699 : REAL;
  INV5_Fan2_Fault_104 AT %QD700 : REAL;
  INV5_Fan3_Fault_104 AT %QD701 : REAL;
  INV5_Fan4_Fault_104 AT %QD702 : REAL;
  INV6_Status_104 AT %QD703 : REAL;  (* *Inverter-6* *)
  INV6_Pin_104 AT %QD704 : REAL;
  INV6_Pv1_voltage_104 AT %QD705 : REAL;
  INV6_Pv1_current_104 AT %QD706 : REAL;
  INV6_Pv1_Pin_104 AT %QD707 : REAL;
  INV6_Pv2_voltage_104 AT %QD708 : REAL;
  INV6_Pv2_current_104 AT %QD709 : REAL;
  INV6_Pv2_Pin_104 AT %QD710 : REAL;
  INV6_Pv3_voltage_104 AT %QD711 : REAL;
  INV6_Pv3_current_104 AT %QD712 : REAL;
  INV6_Pv3_Pin_104 AT %QD713 : REAL;
  INV6_Pv4_voltage_104 AT %QD714 : REAL;
  INV6_Pv4_current_104 AT %QD715 : REAL;
  INV6_Pv4_Pin_104 AT %QD716 : REAL;
  INV6_Pv5_voltage_104 AT %QD717 : REAL;
  INV6_Pv5_current_104 AT %QD718 : REAL;
  INV6_Pv5_Pin_104 AT %QD719 : REAL;
  INV6_Pv6_voltage_104 AT %QD720 : REAL;
  INV6_Pv6_current_104 AT %QD721 : REAL;
  INV6_Pv6_Pin_104 AT %QD722 : REAL;
  INV6_Pv7_voltage_104 AT %QD723 : REAL;
  INV6_Pv7_current_104 AT %QD724 : REAL;
  INV6_Pv7_Pin_104 AT %QD725 : REAL;
  INV6_Pv8_voltage_104 AT %QD726 : REAL;
  INV6_Pv8_current_104 AT %QD727 : REAL;
  INV6_Pv8_Pin_104 AT %QD728 : REAL;
  INV6_Pv9_voltage_104 AT %QD729 : REAL;
  INV6_Pv9_current_104 AT %QD730 : REAL;
  INV6_Pv9_Pin_104 AT %QD731 : REAL;
  INV6_Pv10_voltage_104 AT %QD732 : REAL;
  INV6_Pv10_current_104 AT %QD733 : REAL;
  INV6_Pv10_Pin_104 AT %QD734 : REAL;
  INV6_Pac_out_104 AT %QD735 : REAL;
  INV6_Fac_104 AT %QD736 : REAL;
  INV6_Vac1_104 AT %QD737 : REAL;
  INV6_Iac1_104 AT %QD738 : REAL;
  INV6_Pac1_104 AT %QD739 : REAL;
  INV6_Vac2_104 AT %QD740 : REAL;
  INV6_Iac2_104 AT %QD741 : REAL;
  INV6_Pac2_104 AT %QD742 : REAL;
  INV6_Vac3_104 AT %QD743 : REAL;
  INV6_Iac3_104 AT %QD744 : REAL;
  INV6_Pac3_104 AT %QD745 : REAL;
  INV6_Vac_RS_104 AT %QD746 : REAL;
  INV6_Vac_ST_104 AT %QD747 : REAL;
  INV6_Vac_TR_104 AT %QD748 : REAL;
  INV6_Eactoday_104 AT %QD749 : REAL;
  INV6_Eactotal_104 AT %QD750 : REAL;
  INV6_Timetotal_104 AT %QD751 : REAL;
  INV6_Epv1_today_104 AT %QD752 : REAL;
  INV6_Epv1_total_104 AT %QD753 : REAL;
  INV6_Epv2_today_104 AT %QD754 : REAL;
  INV6_Epv2_total_104 AT %QD755 : REAL;
  INV6_Epv3_today_104 AT %QD756 : REAL;
  INV6_Epv3_total_104 AT %QD757 : REAL;
  INV6_Epv4_today_104 AT %QD758 : REAL;
  INV6_Epv4_total_104 AT %QD759 : REAL;
  INV6_Epv5_today_104 AT %QD760 : REAL;
  INV6_Epv5_total_104 AT %QD761 : REAL;
  INV6_Epv6_today_104 AT %QD762 : REAL;
  INV6_Epv6_total_104 AT %QD763 : REAL;
  INV6_Epv7_today_104 AT %QD764 : REAL;
  INV6_Epv7_total_104 AT %QD765 : REAL;
  INV6_Epv8_today_104 AT %QD766 : REAL;
  INV6_Epv8_total_104 AT %QD767 : REAL;
  INV6_Epv9_today_104 AT %QD768 : REAL;
  INV6_Epv9_total_104 AT %QD769 : REAL;
  INV6_Epv10_today_104 AT %QD770 : REAL;
  INV6_Epv10_total_104 AT %QD771 : REAL;
  INV6_Epv_total_104 AT %QD772 : REAL;
  INV6_Temp1_104 AT %QD773 : REAL;
  INV6_Temp2_104 AT %QD774 : REAL;
  INV6_Temp3_104 AT %QD775 : REAL;
  INV6_Temp4_104 AT %QD776 : REAL;
  INV6_BatVolt_DSP_104 AT %QD777 : REAL;
  INV6_P_Bus_Voltage_104 AT %QD778 : REAL;
  INV6_N_Bus_Voltage_104 AT %QD779 : REAL;
  INV6_IPF_104 AT %QD780 : REAL;
  INV6_String_V1_104 AT %QD781 : REAL;
  INV6_String_I1_104 AT %QD782 : REAL;
  INV6_String_V2_104 AT %QD783 : REAL;
  INV6_String_I2_104 AT %QD784 : REAL;
  INV6_String_V3_104 AT %QD785 : REAL;
  INV6_String_I3_104 AT %QD786 : REAL;
  INV6_String_V4_104 AT %QD787 : REAL;
  INV6_String_I4_104 AT %QD788 : REAL;
  INV6_String_V5_104 AT %QD789 : REAL;
  INV6_String_I5_104 AT %QD790 : REAL;
  INV6_String_V6_104 AT %QD791 : REAL;
  INV6_String_I6_104 AT %QD792 : REAL;
  INV6_String_V7_104 AT %QD793 : REAL;
  INV6_String_I7_104 AT %QD794 : REAL;
  INV6_String_V8_104 AT %QD795 : REAL;
  INV6_String_I8_104 AT %QD796 : REAL;
  INV6_String_V9_104 AT %QD797 : REAL;
  INV6_String_I9_104 AT %QD798 : REAL;
  INV6_String_V10_104 AT %QD799 : REAL;
  INV6_String_I10_104 AT %QD800 : REAL;
  INV6_String_V11_104 AT %QD801 : REAL;
  INV6_String_I11_104 AT %QD802 : REAL;
  INV6_String_V12_104 AT %QD803 : REAL;
  INV6_String_I12_104 AT %QD804 : REAL;
  INV6_String_V13_104 AT %QD805 : REAL;
  INV6_String_I13_104 AT %QD806 : REAL;
  INV6_String_V14_104 AT %QD807 : REAL;
  INV6_String_I14_104 AT %QD808 : REAL;
  INV6_String_V15_104 AT %QD809 : REAL;
  INV6_String_I15_104 AT %QD810 : REAL;
  INV6_String_V16_104 AT %QD811 : REAL;
  INV6_String_I16_104 AT %QD812 : REAL;
  INV6_String_V17_104 AT %QD813 : REAL;
  INV6_String_I17_104 AT %QD814 : REAL;
  INV6_String_V18_104 AT %QD815 : REAL;
  INV6_String_I18_104 AT %QD816 : REAL;
  INV6_String_V19_104 AT %QD817 : REAL;
  INV6_String_I19_104 AT %QD818 : REAL;
  INV6_String_V20_104 AT %QD819 : REAL;
  INV6_String_I20_104 AT %QD820 : REAL;
  INV6_Fan1_Fault_104 AT %QD821 : REAL;
  INV6_Fan2_Fault_104 AT %QD822 : REAL;
  INV6_Fan3_Fault_104 AT %QD823 : REAL;
  INV6_Fan4_Fault_104 AT %QD824 : REAL;
  INV7_Status_104 AT %QD825 : REAL;  (* *Inverter-7* *)
  INV7_Pin_104 AT %QD826 : REAL;
  INV7_Pv1_voltage_104 AT %QD827 : REAL;
  INV7_Pv1_current_104 AT %QD828 : REAL;
  INV7_Pv1_Pin_104 AT %QD829 : REAL;
  INV7_Pv2_voltage_104 AT %QD830 : REAL;
  INV7_Pv2_current_104 AT %QD831 : REAL;
  INV7_Pv2_Pin_104 AT %QD832 : REAL;
  INV7_Pv3_voltage_104 AT %QD833 : REAL;
  INV7_Pv3_current_104 AT %QD834 : REAL;
  INV7_Pv3_Pin_104 AT %QD835 : REAL;
  INV7_Pv4_voltage_104 AT %QD836 : REAL;
  INV7_Pv4_current_104 AT %QD837 : REAL;
  INV7_Pv4_Pin_104 AT %QD838 : REAL;
  INV7_Pv5_voltage_104 AT %QD839 : REAL;
  INV7_Pv5_current_104 AT %QD840 : REAL;
  INV7_Pv5_Pin_104 AT %QD841 : REAL;
  INV7_Pv6_voltage_104 AT %QD842 : REAL;
  INV7_Pv6_current_104 AT %QD843 : REAL;
  INV7_Pv6_Pin_104 AT %QD844 : REAL;
  INV7_Pv7_voltage_104 AT %QD845 : REAL;
  INV7_Pv7_current_104 AT %QD846 : REAL;
  INV7_Pv7_Pin_104 AT %QD847 : REAL;
  INV7_Pv8_voltage_104 AT %QD848 : REAL;
  INV7_Pv8_current_104 AT %QD849 : REAL;
  INV7_Pv8_Pin_104 AT %QD850 : REAL;
  INV7_Pv9_voltage_104 AT %QD851 : REAL;
  INV7_Pv9_current_104 AT %QD852 : REAL;
  INV7_Pv9_Pin_104 AT %QD853 : REAL;
  INV7_Pv10_voltage_104 AT %QD854 : REAL;
  INV7_Pv10_current_104 AT %QD855 : REAL;
  INV7_Pv10_Pin_104 AT %QD856 : REAL;
  INV7_Pac_out_104 AT %QD857 : REAL;
  INV7_Fac_104 AT %QD858 : REAL;
  INV7_Vac1_104 AT %QD859 : REAL;
  INV7_Iac1_104 AT %QD860 : REAL;
  INV7_Pac1_104 AT %QD861 : REAL;
  INV7_Vac2_104 AT %QD862 : REAL;
  INV7_Iac2_104 AT %QD863 : REAL;
  INV7_Pac2_104 AT %QD864 : REAL;
  INV7_Vac3_104 AT %QD865 : REAL;
  INV7_Iac3_104 AT %QD866 : REAL;
  INV7_Pac3_104 AT %QD867 : REAL;
  INV7_Vac_RS_104 AT %QD868 : REAL;
  INV7_Vac_ST_104 AT %QD869 : REAL;
  INV7_Vac_TR_104 AT %QD870 : REAL;
  INV7_Eactoday_104 AT %QD871 : REAL;
  INV7_Eactotal_104 AT %QD872 : REAL;
  INV7_Timetotal_104 AT %QD873 : REAL;
  INV7_Epv1_today_104 AT %QD874 : REAL;
  INV7_Epv1_total_104 AT %QD875 : REAL;
  INV7_Epv2_today_104 AT %QD876 : REAL;
  INV7_Epv2_total_104 AT %QD877 : REAL;
  INV7_Epv3_today_104 AT %QD878 : REAL;
  INV7_Epv3_total_104 AT %QD879 : REAL;
  INV7_Epv4_today_104 AT %QD880 : REAL;
  INV7_Epv4_total_104 AT %QD881 : REAL;
  INV7_Epv5_today_104 AT %QD882 : REAL;
  INV7_Epv5_total_104 AT %QD883 : REAL;
  INV7_Epv6_today_104 AT %QD884 : REAL;
  INV7_Epv6_total_104 AT %QD885 : REAL;
  INV7_Epv7_today_104 AT %QD886 : REAL;
  INV7_Epv7_total_104 AT %QD887 : REAL;
  INV7_Epv8_today_104 AT %QD888 : REAL;
  INV7_Epv8_total_104 AT %QD889 : REAL;
  INV7_Epv9_today_104 AT %QD890 : REAL;
  INV7_Epv9_total_104 AT %QD891 : REAL;
  INV7_Epv10_today_104 AT %QD892 : REAL;
  INV7_Epv10_total_104 AT %QD893 : REAL;
  INV7_Epv_total_104 AT %QD894 : REAL;
  INV7_Temp1_104 AT %QD895 : REAL;
  INV7_Temp2_104 AT %QD896 : REAL;
  INV7_Temp3_104 AT %QD897 : REAL;
  INV7_Temp4_104 AT %QD898 : REAL;
  INV7_BatVolt_DSP_104 AT %QD899 : REAL;
  INV7_P_Bus_Voltage_104 AT %QD900 : REAL;
  INV7_N_Bus_Voltage_104 AT %QD901 : REAL;
  INV7_IPF_104 AT %QD902 : REAL;
  INV7_String_V1_104 AT %QD903 : REAL;
  INV7_String_I1_104 AT %QD904 : REAL;
  INV7_String_V2_104 AT %QD905 : REAL;
  INV7_String_I2_104 AT %QD906 : REAL;
  INV7_String_V3_104 AT %QD907 : REAL;
  INV7_String_I3_104 AT %QD908 : REAL;
  INV7_String_V4_104 AT %QD909 : REAL;
  INV7_String_I4_104 AT %QD910 : REAL;
  INV7_String_V5_104 AT %QD911 : REAL;
  INV7_String_I5_104 AT %QD912 : REAL;
  INV7_String_V6_104 AT %QD913 : REAL;
  INV7_String_I6_104 AT %QD914 : REAL;
  INV7_String_V7_104 AT %QD915 : REAL;
  INV7_String_I7_104 AT %QD916 : REAL;
  INV7_String_V8_104 AT %QD917 : REAL;
  INV7_String_I8_104 AT %QD918 : REAL;
  INV7_String_V9_104 AT %QD919 : REAL;
  INV7_String_I9_104 AT %QD920 : REAL;
  INV7_String_V10_104 AT %QD921 : REAL;
  INV7_String_I10_104 AT %QD922 : REAL;
  INV7_String_V11_104 AT %QD923 : REAL;
  INV7_String_I11_104 AT %QD924 : REAL;
  INV7_String_V12_104 AT %QD925 : REAL;
  INV7_String_I12_104 AT %QD926 : REAL;
  INV7_String_V13_104 AT %QD927 : REAL;
  INV7_String_I13_104 AT %QD928 : REAL;
  INV7_String_V14_104 AT %QD929 : REAL;
  INV7_String_I14_104 AT %QD930 : REAL;
  INV7_String_V15_104 AT %QD931 : REAL;
  INV7_String_I15_104 AT %QD932 : REAL;
  INV7_String_V16_104 AT %QD933 : REAL;
  INV7_String_I16_104 AT %QD934 : REAL;
  INV7_String_V17_104 AT %QD935 : REAL;
  INV7_String_I17_104 AT %QD936 : REAL;
  INV7_String_V18_104 AT %QD937 : REAL;
  INV7_String_I18_104 AT %QD938 : REAL;
  INV7_String_V19_104 AT %QD939 : REAL;
  INV7_String_I19_104 AT %QD940 : REAL;
  INV7_String_V20_104 AT %QD941 : REAL;
  INV7_String_I20_104 AT %QD942 : REAL;
  INV7_Fan1_Fault_104 AT %QD943 : REAL;
  INV7_Fan2_Fault_104 AT %QD944 : REAL;
  INV7_Fan3_Fault_104 AT %QD945 : REAL;
  INV7_Fan4_Fault_104 AT %QD946 : REAL;
  INV8_Status_104 AT %QD947 : REAL;  (* *Inverter-8* *)
  INV8_Pin_104 AT %QD948 : REAL;
  INV8_Pv1_voltage_104 AT %QD949 : REAL;
  INV8_Pv1_current_104 AT %QD950 : REAL;
  INV8_Pv1_Pin_104 AT %QD951 : REAL;
  INV8_Pv2_voltage_104 AT %QD952 : REAL;
  INV8_Pv2_current_104 AT %QD953 : REAL;
  INV8_Pv2_Pin_104 AT %QD954 : REAL;
  INV8_Pv3_voltage_104 AT %QD955 : REAL;
  INV8_Pv3_current_104 AT %QD956 : REAL;
  INV8_Pv3_Pin_104 AT %QD957 : REAL;
  INV8_Pv4_voltage_104 AT %QD958 : REAL;
  INV8_Pv4_current_104 AT %QD959 : REAL;
  INV8_Pv4_Pin_104 AT %QD960 : REAL;
  INV8_Pv5_voltage_104 AT %QD961 : REAL;
  INV8_Pv5_current_104 AT %QD962 : REAL;
  INV8_Pv5_Pin_104 AT %QD963 : REAL;
  INV8_Pv6_voltage_104 AT %QD964 : REAL;
  INV8_Pv6_current_104 AT %QD965 : REAL;
  INV8_Pv6_Pin_104 AT %QD966 : REAL;
  INV8_Pv7_voltage_104 AT %QD967 : REAL;
  INV8_Pv7_current_104 AT %QD968 : REAL;
  INV8_Pv7_Pin_104 AT %QD969 : REAL;
  INV8_Pv8_voltage_104 AT %QD970 : REAL;
  INV8_Pv8_current_104 AT %QD971 : REAL;
  INV8_Pv8_Pin_104 AT %QD972 : REAL;
  INV8_Pv9_voltage_104 AT %QD973 : REAL;
  INV8_Pv9_current_104 AT %QD974 : REAL;
  INV8_Pv9_Pin_104 AT %QD975 : REAL;
  INV8_Pv10_voltage_104 AT %QD976 : REAL;
  INV8_Pv10_current_104 AT %QD977 : REAL;
  INV8_Pv10_Pin_104 AT %QD978 : REAL;
  INV8_Pac_out_104 AT %QD979 : REAL;
  INV8_Fac_104 AT %QD980 : REAL;
  INV8_Vac1_104 AT %QD981 : REAL;
  INV8_Iac1_104 AT %QD982 : REAL;
  INV8_Pac1_104 AT %QD983 : REAL;
  INV8_Vac2_104 AT %QD984 : REAL;
  INV8_Iac2_104 AT %QD985 : REAL;
  INV8_Pac2_104 AT %QD986 : REAL;
  INV8_Vac3_104 AT %QD987 : REAL;
  INV8_Iac3_104 AT %QD988 : REAL;
  INV8_Pac3_104 AT %QD989 : REAL;
  INV8_Vac_RS_104 AT %QD990 : REAL;
  INV8_Vac_ST_104 AT %QD991 : REAL;
  INV8_Vac_TR_104 AT %QD992 : REAL;
  INV8_Eactoday_104 AT %QD993 : REAL;
  INV8_Eactotal_104 AT %QD994 : REAL;
  INV8_Timetotal_104 AT %QD995 : REAL;
  INV8_Epv1_today_104 AT %QD996 : REAL;
  INV8_Epv1_total_104 AT %QD997 : REAL;
  INV8_Epv2_today_104 AT %QD998 : REAL;
  INV8_Epv2_total_104 AT %QD999 : REAL;
  INV8_Epv3_today_104 AT %QD1000 : REAL;
  INV8_Epv3_total_104 AT %QD1001 : REAL;
  INV8_Epv4_today_104 AT %QD1002 : REAL;
  INV8_Epv4_total_104 AT %QD1003 : REAL;
  INV8_Epv5_today_104 AT %QD1004 : REAL;
  INV8_Epv5_total_104 AT %QD1005 : REAL;
  INV8_Epv6_today_104 AT %QD1006 : REAL;
  INV8_Epv6_total_104 AT %QD1007 : REAL;
  INV8_Epv7_today_104 AT %QD1008 : REAL;
  INV8_Epv7_total_104 AT %QD1009 : REAL;
  INV8_Epv8_today_104 AT %QD1010 : REAL;
  INV8_Epv8_total_104 AT %QD1011 : REAL;
  INV8_Epv9_today_104 AT %QD1012 : REAL;
  INV8_Epv9_total_104 AT %QD1013 : REAL;
  INV8_Epv10_today_104 AT %QD1014 : REAL;
  INV8_Epv10_total_104 AT %QD1015 : REAL;
  INV8_Epv_total_104 AT %QD1016 : REAL;
  INV8_Temp1_104 AT %QD1017 : REAL;
  INV8_Temp2_104 AT %QD1018 : REAL;
  INV8_Temp3_104 AT %QD1019 : REAL;
  INV8_Temp4_104 AT %QD1020 : REAL;
  INV8_BatVolt_DSP_104 AT %QD1021 : REAL;
  INV8_P_Bus_Voltage_104 AT %QD1022 : REAL;
  INV8_N_Bus_Voltage_104 AT %QD1023 : REAL;
  INV8_IPF_104 AT %QD1024 : REAL;
  INV8_String_V1_104 AT %QD1025 : REAL;
  INV8_String_I1_104 AT %QD1026 : REAL;
  INV8_String_V2_104 AT %QD1027 : REAL;
  INV8_String_I2_104 AT %QD1028 : REAL;
  INV8_String_V3_104 AT %QD1029 : REAL;
  INV8_String_I3_104 AT %QD1030 : REAL;
  INV8_String_V4_104 AT %QD1031 : REAL;
  INV8_String_I4_104 AT %QD1032 : REAL;
  INV8_String_V5_104 AT %QD1033 : REAL;
  INV8_String_I5_104 AT %QD1034 : REAL;
  INV8_String_V6_104 AT %QD1035 : REAL;
  INV8_String_I6_104 AT %QD1036 : REAL;
  INV8_String_V7_104 AT %QD1037 : REAL;
  INV8_String_I7_104 AT %QD1038 : REAL;
  INV8_String_V8_104 AT %QD1039 : REAL;
  INV8_String_I8_104 AT %QD1040 : REAL;
  INV8_String_V9_104 AT %QD1041 : REAL;
  INV8_String_I9_104 AT %QD1042 : REAL;
  INV8_String_V10_104 AT %QD1043 : REAL;
  INV8_String_I10_104 AT %QD1044 : REAL;
  INV8_String_V11_104 AT %QD1045 : REAL;
  INV8_String_I11_104 AT %QD1046 : REAL;
  INV8_String_V12_104 AT %QD1047 : REAL;
  INV8_String_I12_104 AT %QD1048 : REAL;
  INV8_String_V13_104 AT %QD1049 : REAL;
  INV8_String_I13_104 AT %QD1050 : REAL;
  INV8_String_V14_104 AT %QD1051 : REAL;
  INV8_String_I14_104 AT %QD1052 : REAL;
  INV8_String_V15_104 AT %QD1053 : REAL;
  INV8_String_I15_104 AT %QD1054 : REAL;
  INV8_String_V16_104 AT %QD1055 : REAL;
  INV8_String_I16_104 AT %QD1056 : REAL;
  INV8_String_V17_104 AT %QD1057 : REAL;
  INV8_String_I17_104 AT %QD1058 : REAL;
  INV8_String_V18_104 AT %QD1059 : REAL;
  INV8_String_I18_104 AT %QD1060 : REAL;
  INV8_String_V19_104 AT %QD1061 : REAL;
  INV8_String_I19_104 AT %QD1062 : REAL;
  INV8_String_V20_104 AT %QD1063 : REAL;
  INV8_String_I20_104 AT %QD1064 : REAL;
  INV8_Fan1_Fault_104 AT %QD1065 : REAL;
  INV8_Fan2_Fault_104 AT %QD1066 : REAL;
  INV8_Fan3_Fault_104 AT %QD1067 : REAL;
  INV8_Fan4_Fault_104 AT %QD1068 : REAL;
  Red_Sebeke_Ariza_104 AT %QD1069 : REAL;  (* *Remote_IO* *)
  H1_CB_OPEN_104 AT %QD1070 : REAL;
  H1_CB_CLOSE_104 AT %QD1071 : REAL;
  H1_DS_OPEN_104 AT %QD1072 : REAL;
  H1_DS_CLOSE_104 AT %QD1073 : REAL;
  H1_EDS_OPEN_104 AT %QD1074 : REAL;
  H1_EDS_CLOSE_104 AT %QD1075 : REAL;
  H1_CB_SPRING_104 AT %QD1076 : REAL;
  H1_SF6_LOW_104 AT %QD1077 : REAL;
  H1_SF6_NO_104 AT %QD1078 : REAL;
  H3_CB_OPEN_104 AT %QD1079 : REAL;
  H3_CB_CLOSE_104 AT %QD1080 : REAL;
  H3_TERMOSTAT_TRIP_104 AT %QD1081 : REAL;
  H3_TERMOSTAT_ALARM_104 AT %QD1082 : REAL;
  H4_CB_OPEN_104 AT %QD1083 : REAL;
  H4_CB_CLOSE_104 AT %QD1084 : REAL;
  H4_TERMOSTAT_TRIP_104 AT %QD1085 : REAL;
  H4_TERMOSTAT_ALARM_104 AT %QD1086 : REAL;
  AG_TMS_OPEN_104 AT %QD1087 : REAL;  (* *WAGO I0* *)
  AG_TMS_CLOSE_104 AT %QD1088 : REAL;
  Deprem_Sensor_104 AT %QD1089 : REAL;
  Red_Fault_104 AT %QD1090 : REAL;
  Red_DC_Low_104 AT %QD1091 : REAL;
  Red_AC_Low_104 AT %QD1092 : REAL;
  Red_Aku_Zayif_104 AT %QD1093 : REAL;
  Rtu_Local_Remote_104 AT %QD1094 : REAL;
  Pyronometer_Com_Error AT %QD1095 : REAL;  (* Communication *)
  Refcell1_Com_Error AT %QD1096 : REAL;
  Refcell2_Com_Error AT %QD1097 : REAL;
  H1_Relay_Com_Error AT %QD1098 : REAL;
  H2_EKK_Com_Error AT %QD1099 : REAL;
  INV1_Com_Error AT %QD1100 : REAL;
  INV2_Com_Error AT %QD1101 : REAL;
  INV3_Com_Error AT %QD1102 : REAL;
  INV4_Com_Error AT %QD1103 : REAL;
  INV5_Com_Error AT %QD1104 : REAL;
  INV6_Com_Error AT %QD1105 : REAL;
  INV7_Com_Error AT %QD1106 : REAL;
  INV8_Com_Error AT %QD1107 : REAL;
  Remote_IO_Com_Error AT %QD1108 : REAL;
  TOT_Pin_104 AT %QD1109 : REAL;
  TOT_Com_Error AT %QD1110 : REAL;
  TOT_Eactoday_104 AT %QD1111 : REAL;
  SUM_Non_Com AT %QD1112 : REAL;
  AG_TMS_OPEN_CMD : BOOL;
  AG_TMS_CLOSE_CMD : BOOL;
END_VAR
